# EPICS IOC start-up script: iocsh/filterDrive.iocsh
# ### filterDrive.iocsh ###

#- ###################################################
#- PREFIX           - IOC Prefix
#- INSTANCE         - Instance Prefix
#- KEV              - Name of PV channel giving beam energy in keV.
#- NUM_FILTERS      - Number of filter records loaded in substitutions file
#- SUB              - Optional: Filter settings substitutions file (filterBladeNoSensor.db)
#-                              Macros P and R will be set automatically
#-                    Default: $(OPTICS)/iocsh/EXAMPLE_filterDrive.substitutions
#- OPTICS           - Location of optics module
#- ###################################################

dbLoadTemplate("$(SUB=EXAMPLE_filterDrive.substitutions)", "P=$(PREFIX), R=$(INSTANCE):")
dbLoadRecords("$(OPTICS)/opticsApp/Db/filterDrive.db", "P=$(PREFIX), R=$(INSTANCE):, DESC=Filters, KEV=$(KEV)")
doAfterIocInit("seq filterDrive,'NAME=$(INSTANCE),P=$(PREFIX),R=$(INSTANCE):,NUM_FILTERS=$(NUM_FILTERS)'")
